// TwinCAT 3 PLC project Untitled1
// ProgramVersion: 3.1.4024.0
// libraries:
//   Tc2_Math, * (Beckhoff Automation GmbH)
//   Tc2_Standard, * (Beckhoff Automation GmbH)
//   Tc2_System, * (Beckhoff Automation GmbH)
//   Tc2_Utilities, * (Beckhoff Automation GmbH)
//   Tc3_CM, * (Beckhoff Automation GmbH)
//   Tc3_CM_Base, * (Beckhoff Automation GmbH)
//   Tc3_IotBase, * (Beckhoff Automation GmbH)
//   Tc3_JsonXml, * (Beckhoff Automation GmbH)
//   Tc3_Module, * (Beckhoff Automation GmbH)
//   Tc3_MultiArray, * (Beckhoff Automation GmbH)
// project tree:
//   / CM_Process_Task.TcTTO, HTTP_Task.TcTTO, PlcTask.TcTTO
//   DUTs/Error Monitoring/ ST_HRErrHist.TcDUT, E_TalkToGateway_Err.TcDUT
//   DUTs/ E_AnalysisIDs.TcDUT, E_IsoClass.TcDUT, E_RequestType.TcTLEO, ST_ReceivedData.TcDUT
//   DUTs/Function Generator/ E_FunctionType.TcDUT
//   FUBs/ FB_Flash.TcPOU, FB_FunctionGenerator.TcPOU, FB_FunctionGenerator_1.TcPOU, FB_HRErrHist.TcPOU
//   GVLs/ GLOBAL.TcGVL, GVL_Const.TcGVL
//   POUs/CM_Collection/ CM_SensorWorks_Sensor1.TcPOU, CM_SensorWorks_Sensor2.TcPOU, CM_Sim.TcPOU
//   POUs/CM_Processing/ CM_SensorWorks_Sensor1ISO.TcPOU, CM_SensorWorks_Sensor2ISO.TcPOU, CM_Sim_ISO.TcPOU
//   POUs/HTTP/ FB_RequestToGateway.TcPOU, FB_TalkToGateway.TcPOU, GetDataFromSensorWorksHTTP.TcPOU
//   POUs/ MAIN.TcPOU
// real-time tasks:
//   TASK PlcTask: cycle T#25000us, priority 10, ADS port 350
//   TASK CM_Process_Task: cycle T#50000us, priority 4, ADS port 351
//   TASK HTTP_Task: cycle T#500ms, priority 20, ADS port 352

CONFIGURATION Untitled1
    RESOURCE PLC ON TwinCAT3
        TASK CM_Process_Task(INTERVAL := T#50000us, PRIORITY := 4);
        TASK HTTP_Task(INTERVAL := T#500ms, PRIORITY := 20);
        TASK PlcTask(INTERVAL := T#25000us, PRIORITY := 10);
        PROGRAM CM_Sim_ISO WITH CM_Process_Task : CM_Sim_ISO;
        PROGRAM CM_SensorWorks_Sensor1ISO WITH CM_Process_Task : CM_SensorWorks_Sensor1ISO;
        PROGRAM CM_SensorWorks_Sensor2ISO WITH CM_Process_Task : CM_SensorWorks_Sensor2ISO;
        PROGRAM MAIN WITH PlcTask : MAIN;
    END_RESOURCE
END_CONFIGURATION

// ---- DUTs/Error Monitoring/ST_HRErrHist.TcDUT
TYPE ST_HRErrHist :
STRUCT
{attribute 'displaymode':='hex'}
	hrErrCode	: HRESULT;
	sErrSource	: STRING(63);
	nErrCount	: UDINT;
END_STRUCT
END_TYPE

// ---- DUTs/Error Monitoring/E_TalkToGateway_Err.TcDUT

TYPE
    E_TalkToGateway_Err :
    (
        e_NoIPAddress           := 10,
        e_NoPortNumber          := 20,
        e_NoDeviceID            := 30,
        e_DeviceIDOutsideLimits := 31,
        e_DeviceIDNotFound      := 32,
		e_JSONRequestError		:= 40
        );
END_TYPE

// ---- DUTs/E_AnalysisIDs.TcDUT
TYPE
    E_AnalysisIDs :
    (
        (* analysis chain *)
        eID_SimSource := 1,
        eID_SimISO,
        eID_SimSinkISO,
        eID_SimSpectrumCh1,
        eID_SimSpectrumCh2,
        eID_SimSinkSpectrumCh1,
        eID_SimSinkSpectrumCh2,
        eID_SensorWorksSource,
        eID_SensorWorksISO,
        eID_SensorWorksSpectrum,
        eID_SensorWorksSinkISO,
        eID_SensorWorkSinkSpectrum,
        eID_SW_Source_Device_1,
        eID_SW_ISO_Device_1,
        eID_SW_Sink_Device_1,
        eID_SW_Source_Device_2,
        eID_SW_ISO_Device_2,
        eID_SW_Sink_Device_2
    ) UDINT;
END_TYPE

// ---- DUTs/E_IsoClass.TcDUT
(* ISO Classes *)
{attribute 'qualified_only'}
TYPE E_IsoClass :
(
	A := 1,
	B,
	C,
	D
) UDINT;
END_TYPE

// ---- DUTs/E_RequestType.TcTLEO

TYPE E_RequestType :
(
	eIdle,
	eSampleRate,
	eTraceLen,
	eMode,
	eRequestSend,
	eViewRequest, // ✅ Add this line
	eGetData,
	eProcess,
	eERROR
);
END_TYPE

// ---- DUTs/Function Generator/E_FunctionType.TcDUT
{attribute 'qualified_only'}
TYPE E_FunctionType :
(
	Sine,		// typical for vibrations originating from rotating machine
	Square,		// mixed sine signals good for analyzing spectrum
	Pulse,		// mixed sine signals good for analyzing spectrum
	Triangular,	// mixed sine signals good for analyzing spectrum
	Sawtooth,	// ramp-type vibrations, continuously increasing
	AM			// amplitude modulation: typical for vibrations originating from gear-tooth failure or bearing faults
);
END_TYPE

// ---- DUTs/ST_ReceivedData.TcDUT
TYPE ST_ReceivedData :
STRUCT
	uuid			: STRING;
	blename			: STRING;
	name			: STRING;
	id				: STRING;
	timestamp		: STRING;
	value 			: ARRAY[0..512] OF DINT;
	value_y			: ARRAY[0..512] OF DINT;
	value_z			: ARRAY[0..512] OF DINT;
	rate			: DINT;
	trace			: DINT;
	count			: DINT;
	gain			: DINT;
	calibration		: LREAL;
	calibration_y	: LREAL;
	calibration_z	: LREAL;
	temperature		: LREAL;
	battery			: LREAL;
	axes			: LREAL;
	mux_axis		: LREAL;
	measured_rate	: LREAL;
	
END_STRUCT
END_TYPE

// ---- GVLs/GLOBAL.TcGVL
{attribute 'qualified_only'}
VAR_GLOBAL
    {attribute 'TcAnalytics'}
    aSimBuffer : ARRAY[1..GVL_Const.cChannels] OF ARRAY[1..GVL_Const.cOversamples] OF LREAL;
    aSimRMSResult         : ARRAY[1..GVL_Const.cChannels] OF ARRAY[1..GVL_Const.cResult_Length] OF LREAL;
    aSimSpectrumCh1Result : ARRAY[1..(GVL_Const.cFFTLength / 2 + 1)] OF LREAL;
    aSimSpectrumCh2Result : ARRAY[1..(GVL_Const.cFFTLength / 2 + 1)] OF LREAL;

	(****** Sensor Works ******)
    stSensorWorksHTTPSensorData : ARRAY[1..GVL_Const.cMaxVibrationDevices] OF ST_ReceivedData; // Data from the devices
    aSensorWorksHTTPInput    : ARRAY[1..GVL_Const.cMaxVibrationDevices] OF ARRAY[1..GVL_Const.cSensorPacket] OF LREAL; // Scaled data to input into vibration FuBs
    aSensorWorkISOHTTPResult : ARRAY[1..GVL_Const.cMaxVibrationDevices] OF ARRAY[1..GVL_Const.cResult_Length] OF LREAL; // Output values from Sink

    strTimeStamp : STRING;
    strIPAddress : STRING := '192.168.4.44';
	//strIPAddress : STRING := '192.168.216.148';
	//strDeviceID  : ARRAY[1..GVL_Const.cMaxVibrationDevices] OF STRING := ['d5:d0:f9:30:83:d7'];
	
	strDeviceID  : ARRAY[1..GVL_Const.cMaxVibrationDevices] OF STRING := ['fa:e2:ad:e2:8d:99', 'd5:d0:f9:30:83:d7'];
    nPortNumber  : UINT := 8080;
	
	bCommError : BOOL := FALSE;     // Qin
//	fbCommErrHist : FB_ErrHist;
    bIsProcessingRequest : BOOL := FALSE;
    strLastRequestOutput : STRING(255);
	
	iAnalueIn1 AT %I* : INT;  // Qin
	Sensor1Ch1AccRMSiAnalueIn2 AT %I* : INT;
	
Sensor1Ch1AccRMS : ARRAY[1..28] OF REAL := [
    37.0, 15.0, 10.0, 23.0, 17.0, 21.0, 23.0, 17.0,
    24.0, 18.0, 3.0, 18.0, 38.0, 29.0, 11.0, 0.0,
    7.0, 20.0, 8.0, 7.0, 24.0, 9.0, 1.0, 28.0,
    29.0, 19.0, 30.0, 28.0
];




END_VAR

// ---- GVLs/GVL_Const.TcGVL
{attribute 'qualified_only'}
VAR_GLOBAL CONSTANT

    cFSample      : UDINT := 10000; // 1ms task with 10 oversamples = 10kHz
    cMaxBins      : UDINT := 100;
    cMaxQuantiles : UDINT := 2;
    cMaxClasses   : UDINT := 3; // Normal, Warning, Alarm		

    // define frequency interval according to ISO 10816-3
    // e.g. 10 .. 1000 Hz for rotating speed over 600r/min
    cfLowerFrequencyLimit : UDINT := 10;
    cfUpperFrequencyLimit : UDINT := 1000;

    // Parameters for RMS calculation
    cOrderRMS      : UDINT := 2;             // ISO 10816-3 requires velocity and displacement, if measured using accelerometer we need to integrate 2 times
    cChannels      : UDINT := 2;             // ISO 10816-3 says 2 orthogonal sensors per measurement location-> 2 channels
    cResult_Length : UDINT := cOrderRMS + 1; // nOrder+1
    cSensorSampleChannels
        : UDINT := 1;

    // Classes according to ISO:
    // machine, elasticty, value
    cISOClassDef_Velocity : ARRAY[1..2, 1..2, 1..3] OF LREAL := [0.0023,
                                                                 0.0045,
                                                                 0.0071,
                                                                 0.0035,
                                                                 0.0071,
                                                                 0.011,
                                                                 0.0014,
                                                                 0.0028,
                                                                 0.0045,
                                                                 0.0023,
                                                                 0.0045,
                                                                 0.0071];
    cISOClassDef_Displ : ARRAY[1..2, 1..2, 1..3] OF LREAL := [2.9E-05,
                                                              5.7E-05,
                                                              9E-05,
                                                              4.5E-05,
                                                              9E-05,
                                                              0.00014,
                                                              2.2E-05,
                                                              4.5E-05,
                                                              7.1E-05,
                                                              3.7E-05,
                                                              7.1E-05,
                                                              0.000113];

    // optional constants if real sensors are applied
    cGravitationalAcc : LREAL := 9.81;  // 1 g approx 9.81 m/s^2 -> physical constant
    cSensitivity      : LREAL := 0.01;  // [in Volts/g] depends on sensor used in application, e.g. 10 mV/g
    cMeasurementRange : LREAL := 5;     // +-5 Volts (EL3632)
    cResolution       : LREAL := 32768; // 2^15 (15 bits resolution + 1 bit sign) (EL3632)
    cScale            : LREAL := cMeasurementRange * cGravitationalAcc / (cSensitivity * cResolution);

    // Application ConMon constants
    cSensorPacket          : UDINT                 := 512; // Number of samples in the packet incoming from the sensor	
    cSensorSampleRate      : UDINT                 := 256;
    cOversamples           : UDINT                 := 10;                             // number of oversamples
    cMaxChannels           : UDINT                 := 5;                              // number of data channels
    cWindowType            : E_CM_WindowType       := E_CM_WindowType.eCM_HannWindow; // window type for analysis
    cWindowParameters      : T_CM_WindowParameters := [0, 0, 0, 0, 0];                // window parameters
    cWindowLength          : UDINT                 := 3200;                           // length of signal window 
    cOverlap               : UDINT                 := 1600;                           // recommended buffer overlap
    cBufferLength          : UDINT                 := cWindowLength - cOverlap;       // internal buffer size with 50% overlapping	                                            						
    cFFTLength             : UDINT                 := 4096;                           // length of FFT for mag. spectrum
    cFFTResult             : UDINT                 := 2049;                           // result of mag. spectrum (cFFTLength/2+1)
    cBufferLength_Spectrum : UDINT                 := 1600;                           // buffer size due to 50% overlap

    //Alarm Constants
    cMax_Alarms : UINT := 99;

    // Device Constants
    cMaxVibrationDevices : UINT := 10;

END_VAR

// ---- POUs/CM_Processing/CM_Sim_ISO.TcPOU
PROGRAM CM_Sim_ISO
VAR CONSTANT
		cInitIntRMS 	: ST_CM_IntegratedRMS_InitPars   := (	nFFT_Length := GVL_Const.cFFTLength, 
															nWindowLength := GVL_Const.cWindowLength,
															fSampleRate := GVL_Const.cFSample,
		 													fLowerFrequencyLimit := GVL_Const.cfLowerFrequencyLimit,
															fUpperFrequencyLimit := GVL_Const.cfUpperFrequencyLimit,
															nOrder := GVL_Const.cOrderRMS,
															nChannels := GVL_Const.cChannels,                        
															eWindowType := E_CM_WindowType.eCM_HannWindow, 
															bTransformToDecibel:= FALSE);		

END_VAR
VAR
		fbRMS				: FB_CMA_IntegratedRMS  	  :=(	stInitPars := cInitIntRMS, 
															nOwnID := eID_SimISO, 
															aDestIDs := [eID_SimSinkISO] );

	fbErrHist			: FB_HRErrHist; // error monitoring


END_VAR

// Call RMS
fbRMS.Call();

IF fbRMS.bError THEN
	fbErrHist.AddError(bErr:=TRUE, hrErrCode:=fbRMS.hrErrorCode, sErrSource:='CM_Sim_ISO.fbRMS'); // error monitoring
	// ToDo: if error
END_IF

END_PROGRAM

// ---- FUBs/FB_HRErrHist.TcPOU
FUNCTION_BLOCK FB_HRErrHist
(* v1.10
build up an error history consisting of two arrays and one index.
The index shows the actual array position. The last error id and the count for this id are saved in the arrays.
If an error id is the same as the previous input error the counter is increased. Otherwise the index is increased.
*)
VAR_INPUT
	bEdgeDetect	: BOOL;	(* FALSE: every input(bErr) is processed; TRUE: only rising edge of input is processed *)
END_VAR
VAR_OUTPUT
	nErrSum		: UINT;
	nErrIdx		: UINT; // error list index of last occured error (max. cHistLen)
	aErrList	: ARRAY[1..cHistLen] OF ST_HRErrHist;
END_VAR

VAR
	bNewErr		: BOOL;
	fbErrTrig	: R_TRIG;
END_VAR
VAR CONSTANT
	cHistLen	: UINT := 100;
END_VAR

METHOD AddError
VAR_INPUT
	bErr		: BOOL;
	hrErrCode	: HRESULT;
	sErrSource	: STRING(63);
END_VAR
fbErrTrig(CLK:=bErr);
IF bEdgeDetect THEN
	bNewErr := fbErrTrig.Q;
ELSE
	bNewErr := bErr;
END_IF

IF bNewErr THEN
	nErrSum := nErrSum + 1;
	IF nErrIdx < cHistLen THEN
		IF nErrIdx = 0 THEN
			nErrIdx	:= nErrIdx + 1;
		ELSIF aErrList[nErrIdx].hrErrCode <> hrErrCode OR aErrList[nErrIdx].sErrSource <> sErrSource THEN
			nErrIdx	:= nErrIdx + 1;
		END_IF
		aErrList[nErrIdx].hrErrCode := hrErrCode;
		aErrList[nErrIdx].sErrSource := sErrSource;
		aErrList[nErrIdx].nErrCount := aErrList[nErrIdx].nErrCount + 1;
	END_IF
END_IF
END_METHOD

METHOD Reset
VAR_INPUT
END_VAR
nErrSum := 0;
nErrIdx := 0;
MEMSET(ADR(aErrList),0,SIZEOF(aErrList));
END_METHOD

END_FUNCTION_BLOCK

// ---- POUs/CM_Processing/CM_SensorWorks_Sensor1ISO.TcPOU
PROGRAM CM_SensorWorks_Sensor1ISO

VAR CONSTANT
		cInitIntRMS 	: ST_CM_IntegratedRMS_InitPars   := (	nFFT_Length := GVL_Const.cSensorPacket, 
															nWindowLength := GVL_Const.cSensorPacket,
															fSampleRate := GVL_Const.cSensorSampleRate, // packets per second, sample time is 2s
		 													fLowerFrequencyLimit := 10,
															fUpperFrequencyLimit := 100,	// needs to be less than half of the sample rate
															nMaxBands:= 1, 										
															nOrder := 2,
															nChannels := 1,                        
															eWindowType := E_CM_WindowType.eCM_HannWindow,
															nOverlap:= 0, 
															bTransformToDecibel:= FALSE);

END_VAR

VAR
	fbRMS				: FB_CMA_IntegratedRMS  	  :=(	stInitPars := cInitIntRMS, 
															nOwnID := eID_SW_ISO_Device_1, 
															aDestIDs := [eID_SW_Sink_Device_1],
															nResultBuffers:= 4);
	
	bInit: BOOL := TRUE;														
	aBands				: ARRAY [1..2] OF LREAL := [10.0, 100.0];
	hResInit			:  HRESULT;										

	fbErrHist			: FB_HRErrHist; // error monitoring

END_VAR

IF bInit THEN
	hResInit := fbRms.Configure(pArg:= ADR(aBands), nArgSize:= SIZEOF(aBands));
	bInit := FALSE;
END_IF

// Call RMS
fbRMS.Call();

IF fbRMS.bError THEN
	fbErrHist.AddError(bErr:=TRUE, hrErrCode:=fbRMS.hrErrorCode, sErrSource:='CM_SensorWorks_Sensor1ISO.fbRMS'); // error monitoring
	// ToDo: if error
END_IF

END_PROGRAM

// ---- POUs/CM_Processing/CM_SensorWorks_Sensor2ISO.TcPOU
PROGRAM CM_SensorWorks_Sensor2ISO

VAR CONSTANT
    cInitIntRMS : ST_CM_IntegratedRMS_InitPars := (nFFT_Length          := GVL_Const.cSensorPacket,
                                                   nWindowLength        := GVL_Const.cSensorPacket,
                                                   fSampleRate          := GVL_Const.cSensorSampleRate, // packets per second, sample time is 2s
                                                   fLowerFrequencyLimit := 10,
                                                   fUpperFrequencyLimit := 100, // needs to be less than half of the sample rate
                                                   nMaxBands            := 1,
                                                   nOrder               := 2,
                                                   nChannels            := 1,
                                                   eWindowType          := E_CM_WindowType.eCM_HannWindow,
                                                   nOverlap             := 0,
                                                   bTransformToDecibel  := FALSE);

END_VAR

VAR
    fbRMS : FB_CMA_IntegratedRMS := (stInitPars     := cInitIntRMS,
                                     nOwnID         := eID_SW_ISO_Device_2,
                                     aDestIDs       := [eID_SW_Sink_Device_2],
                                     nResultBuffers := 4);

    bInit    : BOOL                 := TRUE;
    aBands   : ARRAY[1..2] OF LREAL := [10.0, 100.0];
    hResInit : HRESULT;

    fbErrHist : FB_HRErrHist; // error monitoring

END_VAR

IF bInit THEN
    hResInit := fbRms.Configure(pArg := ADR(aBands), nArgSize := SIZEOF(aBands));
    bInit    := FALSE;
END_IF

// Call RMS
fbRMS.Call();

IF fbRMS.bError THEN
    fbErrHist.AddError(bErr := TRUE, hrErrCode := fbRMS.hrErrorCode, sErrSource := 'CM_SensorWorks_Sensor2ISO.fbRMS'); // error monitoring
    // ToDo: if error
END_IF

END_PROGRAM

// ---- POUs/MAIN.TcPOU
PROGRAM MAIN
VAR
	// Task Vars
	nChannel: UDINT;
	fbFunctionGenerator1	: FB_FunctionGenerator;		// Signal Generator, ch1
	fbFunctionGenerator2	: FB_FunctionGenerator;		// Signal Generator, ch2
	fSetFrequency1			: LREAL := 400;		        // Hz
	fSetAmplitude1			: LREAL := 4;		        // peak amplitude of sin signal [m/s^2]
	fSetFrequency2			: LREAL := 35;		        // Hz
	fSetAmplitude2			: LREAL := 4;		        // peak amplitude of sin signal	[m/s^2]	
	
	bAddDisturbance			: BOOL;											// add fault
	fbDisturbance1			: FB_FunctionGenerator;							// fault simulator
	fDistAmplitude1			: LREAL	:= 5;									// fault amplitude
	fDistFrequency1			: LREAL	:= 200;									// fault frequency (recurring)
	fbDisturbance2			: FB_FunctionGenerator;							// fault simulator
	fDistAmplitude2			: LREAL	:= 2;									// fault amplitude
	fDistFrequency2			: LREAL	:= 100;									// fault frequency (recurring)

	eDistFunction			: E_FunctionType :=  E_FunctionType.Square;	// fault shape
	aDisturbance			: ARRAY[1..GVL_Const.cChannels] OF ARRAY[1..GVL_Const.cOversamples] OF LREAL;

	fbRand					: DRAND;				 	
	fRandomNumber			: LREAL;	
	fVar					: LREAL := 0.38;

	nSample					: UDINT;

	fbTalkToGateway			: FB_TalkToGateway;

END_VAR

VAR   //Qin
    fbSendEdge : R_TRIG;

    bTriggerSend : BOOL := FALSE;
    bStartPulse  : BOOL := TRUE;

    fbHttpClient : FB_IotHttpClient;

   // strRawJson : STRING(8191);

    bBusy   : BOOL;
    bError  : BOOL;
END_VAR


// Simulated frequency generation
fbFunctionGenerator1(fFrequency := fSetFrequency1,
                     fAmplitude := fSetAmplitude1,
                     eFunction  := E_FunctionType.Sine,
                     aSignal    := GLOBAL.aSimBuffer[1]);

fbFunctionGenerator2(fFrequency := fSetFrequency2,
                     fAmplitude := fSetAmplitude2,
                     eFunction  := E_FunctionType.Sine,
                     aSignal    := GLOBAL.aSimBuffer[2]);

IF bAddDisturbance THEN
    // Random number generator
    fbRand(Seed := 1000, Num => fRandomNumber);
    (* Disturbance signal *)
    fbDisturbance1(bEnable    := TRUE,
                   fAmplitude := fDistAmplitude1,
                   fFrequency := fDistFrequency1,
                   fOffset    := 0,
                   nDutyCycle := 2,
                   eFunction  := eDistFunction,
                   aSignal    := aDisturbance[1]);

    fbDisturbance2(bEnable    := TRUE,
                   fAmplitude := fDistAmplitude2,
                   fFrequency := fDistFrequency2,
                   fOffset    := 0,
                   nDutyCycle := 2,
                   eFunction  := eDistFunction,
                   aSignal    := aDisturbance[2]);

    FOR nChannel := 1 TO GVL_Const.cChannels DO
        // Input signal with disturbance
        FOR nSample := 1 TO GVL_Const.cOversamples DO
            GLOBAL.aSimBuffer[nChannel][nSample] := GLOBAL.aSimBuffer[nChannel][nSample] + fRandomNumber * aDisturbance[nChannel][nSample];
        END_FOR
    END_FOR

END_IF

// Statically writing devices for ease during testing
//GLOBAL.strDeviceID[1] := 'e0:f6:fd:c4:e3:08';
//GLOBAL.strDeviceID[2] := 'd5:d0:f9:30:83:d7';

// Instance call to FB_TalkToGateway
fbTalkToGateway(
    strIPAddress        := GLOBAL.strIPAddress,
    nPortNumber         := GLOBAL.nPortNumber,
    strDeviceID         := GLOBAL.strDeviceID,
    bStopConnection     :=,                                  // TODO: Set logic to stop the connection when needed.  
    bResetError         := FALSE,                                  // TODO: Link to a button or watchdog to reset error
    bSendRequest        := ,                                   // Should be controlled by a trigger condition
    eRequestType := E_RequestType.eViewRequest,
	//eRequestType        := E_RequestType.eGetData,              // Replace with actual enum value as needed
    iRequestDeviceIndex := 1,                                      // Index of the device to talk to (1 or 2)
    tPollTime           := T#1S,
    bError              => GLOBAL.bCommError,                      // Assign your error flag
//    fbErrHist           => GLOBAL.fbCommErrHist,                   // Optional: instantiate this function block globally
    aDeviceResponse     => GLOBAL.stSensorWorksHTTPSensorData,    // Structure to receive sensor data
    strRequestOutput    => GLOBAL.strLastRequestOutput,           // Optional: use to log or debug request payloads
    bProcessingRequest  => GLOBAL.bIsProcessingRequest            // Track request state
);


// this block Qin
IF bStartPulse THEN
    bTriggerSend := TRUE;
    bStartPulse := FALSE;
ELSE
    bTriggerSend := FALSE;
END_IF


// Detect rising edge
fbSendEdge(CLK := bTriggerSend);

// Call your FB   //Qin
(*
fbGetDataFromSensor(
    bSend := fbSendEdge.Q,
    strRequest := '/device/d5:d0:f9:30:83:d7/cache/latest',   // Qin
    bErrorReset := FALSE,
    fbClient := fbHttpClient,
    bBusy => bBusy,
    bError => bError
);
*)

// View raw content
// strRawJson := fbGetDataFromSensor.sContent;   //Qin


// Cyclic Program Calls
CM_Sim();
CM_SensorWorks_Sensor1();
CM_SensorWorks_Sensor2();

END_PROGRAM

// ---- FUBs/FB_FunctionGenerator.TcPOU
// generates a signal build up by the specified function type. v1.6
FUNCTION_BLOCK FB_FunctionGenerator
VAR_INPUT
	bEnable		: BOOL 	:= TRUE;	// set TRUE to generate the specified signal; set FALSE to reset the signal buffer
	fFrequency	: LREAL := 1000;	// in [Hz]
	fAmplitude	: LREAL := 1;
	fOffset		: LREAL	:= 0;	
	nDutyCycle	: UINT 	:= 50;		// in [%] (for pulse function)
	eFunction	: E_FunctionType := E_FunctionType.Sine;	
END_VAR
VAR_IN_OUT
	aSignal		: ARRAY[1..GVL_Const.cOversamples] OF LREAL;
END_VAR
VAR_OUTPUT
	bError		: BOOL;
END_VAR

VAR
	bInit						: BOOL := TRUE;
	fbGetTaskIdx				: GETCURTASKINDEX;
	
	fLastFrequency				: LREAL;		// in [Hz]
	fLastAmplitude				: LREAL;
	fLastOffset					: LREAL;
	nLastDutyCycle				: UINT;
	eLastFunction				: E_FunctionType;
	
	nSamples					: UDINT;
	fCycleTime					: LREAL;		// in [s]
	fDelta						: LREAL;		// amplitude delta per sample
	fPhase						: LREAL;		// in [°]
	nSign						: INT := 1;		// 1 or -1
	fLastSignalValue			: LREAL;		// amplitude
	fPeriod						: LREAL;		// in [s]
	fAngularIncrement			: LREAL;		// in [°]
	fAngularIncrementPerCycle	: LREAL;		// in [°]
	fAngularIncrementPerSample	: LREAL;		// in [°]
	(* for modulated signal (carrier signal without offset) *)
	fCarrierFrequency					: LREAL := 500;	// in [Hz] (sine)
	fCarrierAmplitude					: LREAL := 1;
	fCarrierPeriod						: LREAL;		// in [s]
	fCarrierAngularIncrement			: LREAL;		// in [°]
	fCarrierAngularIncrementPerCycle	: LREAL;		// in [°]
	fCarrierAngularIncrementPerSample	: LREAL;		// in [°]
				
END_VAR

IF bEnable THEN
	IF fLastFrequency <> fFrequency THEN
		bInit := TRUE; // For automatic initializing
		fLastFrequency := fFrequency;
	END_IF
	IF fLastAmplitude <> fAmplitude THEN
		bInit := TRUE; // For automatic initializing
		fLastAmplitude := fAmplitude;
	END_IF
	IF fLastOffset <> fOffset THEN
		bInit := TRUE; // For automatic initializing
		fLastOffset := fOffset;
	END_IF
	IF nLastDutyCycle <> nDutyCycle THEN
		bInit := TRUE; // For automatic initializing
		nLastDutyCycle := nDutyCycle;
	END_IF
	IF eLastFunction <> eFunction THEN
		bInit := TRUE; // For automatic initializing
		eLastFunction := eFunction;
	END_IF
	IF bInit THEN
		// Get task info	
		fbGetTaskIdx();
		fCycleTime := UDINT_TO_LREAL(TwinCAT_SystemInfoVarList._TaskInfo[fbGetTaskIdx.index].CycleTime) (*100ns*) / (10.0 * 1000.0 * 1000.0);	
		fLastSignalValue := 0;
		nSign := 1;
		fAngularIncrement := 0;
		// Flush out old data
		MEMSET(ADR(aSignal), 0, SIZEOF(aSignal));
		IF fFrequency > 0 AND fCycleTime > 0 THEN		
			// Calculate period, increments per plc cycle, increment per oversample
			IF GVL_Const.cOversamples > 0 THEN			
				IF eFunction = E_FunctionType.Sine THEN
					fPeriod := 1/fFrequency;
					fAngularIncrementPerCycle := 360*(fCycleTime/fPeriod);
					fAngularIncrementPerSample := fAngularIncrementPerCycle/GVL_Const.cOversamples;
					// no phase adjustment
					bInit := FALSE;	
				ELSIF eFunction = E_FunctionType.Square	THEN
					fPeriod := 1/fFrequency;
					fAngularIncrementPerCycle  := 360*(fCycleTime/fPeriod);
					fAngularIncrementPerSample := fAngularIncrementPerCycle/GVL_Const.cOversamples;
					fPhase := 0.5*360;
					bInit := FALSE;
				ELSIF eFunction = E_FunctionType.Pulse THEN
					fPeriod := 1/fFrequency;
					fAngularIncrementPerCycle  := 360*(fCycleTime/fPeriod);
					fAngularIncrementPerSample := fAngularIncrementPerCycle/GVL_Const.cOversamples;
					IF nDutyCycle > 100 THEN
						nDutyCycle := 100;
					END_IF
					fPhase := (UDINT_TO_LREAL(nDutyCycle)/100)*360;
					bInit := FALSE;					
				ELSIF eFunction = E_FunctionType.Triangular THEN
					fPeriod := 1/fFrequency;				
					fAngularIncrementPerCycle  := 360*(fCycleTime/fPeriod);
					fAngularIncrementPerSample := fAngularIncrementPerCycle/GVL_Const.cOversamples;
					fPhase := 0.5*360; 
					fDelta := 4*(fAmplitude/(360/fAngularIncrementPerSample));				
					bInit := FALSE;
				ELSIF eFunction = E_FunctionType.Sawtooth THEN
					fPeriod := 1/fFrequency;			
					fAngularIncrementPerCycle  := 360*(fCycleTime/fPeriod);		
					fAngularIncrementPerSample := fAngularIncrementPerCycle/GVL_Const.cOversamples;
					fDelta := fAmplitude/(360/fAngularIncrementPerSample);
					bInit := FALSE;
				ELSIF eFunction = E_FunctionType.AM THEN
					fPeriod := 1/fFrequency;
					fAngularIncrementPerCycle := 360*(fCycleTime/fPeriod);
					fAngularIncrementPerSample := fAngularIncrementPerCycle/GVL_Const.cOversamples;
					// no phase adjustment
					fCarrierPeriod := 1/fCarrierFrequency;
					fCarrierAngularIncrementPerCycle := 360*(fCycleTime/fCarrierPeriod);
					fCarrierAngularIncrementPerSample := fCarrierAngularIncrementPerCycle/GVL_Const.cOversamples;				
					// no phase adjustment	
					bInit := FALSE;
				ELSE
					bError := TRUE;	
				END_IF
			ELSE
				bError := TRUE;
			END_IF
		ELSE
			bError := TRUE;
		END_IF
	END_IF
	
	// Enable function generator
	IF NOT bError THEN		
		CASE eFunction OF		
			// sine: typical for vibrations originating from rotating machine
			E_FunctionType.Sine: Sine();
			
			// square: mixed sine signals good for analyzing spectrum				
			E_FunctionType.Square: Square();
			
			// pulse: mixed sine signals good for analyzing spectrum				
			E_FunctionType.Pulse: Pulse();
	
			// sawtooth: ramp-type vibrations, continuously increasing			
			E_FunctionType.Sawtooth: Sawtooth();
		
			// triangular: mixed sine signals good for analyzing spectrum
			E_FunctionType.Triangular: Triangular();
		
			// amplitude modulation: typical for vibrations originating from gear-tooth failure or bearing faults
			// Carrier signal with own frequency and amplitude		
			E_FunctionType.AM: AM();				
		END_CASE
	END_IF
ELSE
	// Flush out old data
	MEMSET(ADR(aSignal), 0, SIZEOF(aSignal));
	
	bInit := TRUE;
	bError := FALSE;
END_IF

METHOD PRIVATE AM
VAR_INPUT
END_VAR
{warning disable C0371}

FOR nSamples := 1 TO GVL_Const.cOversamples DO
	// base signal * carrier signal
	aSignal[nSamples] := ( fAmplitude*SIN(2*PI*(fAngularIncrement+(nSamples-1)*fAngularIncrementPerSample)/360) + fOffset )
							* ( fCarrierAmplitude*SIN(2*PI*(fCarrierAngularIncrement+(nSamples-1)*fCarrierAngularIncrementPerSample)/360) );
END_FOR
// Increment angular positions
fAngularIncrement := fAngularIncrement + fAngularIncrementPerCycle;
fCarrierAngularIncrement := fCarrierAngularIncrement + fCarrierAngularIncrementPerCycle;

{warning restore C0371}
END_METHOD

METHOD PRIVATE Pulse
VAR_INPUT
END_VAR
{warning disable C0371}

FOR nSamples := 1 TO GVL_Const.cOversamples DO
	// For pulse wave (unequal phases)
	IF (fAngularIncrement >= 360) THEN
		fAngularIncrement := fAngularIncrement - DINT_TO_LREAL(LREAL_TO_DINT(fAngularIncrement/360))*360;
		// or with Tc2_Math library: fAngularIncrement := LMOD(fAngularIncrement,360);
	END_IF
	IF (fAngularIncrement < fPhase) THEN
		nSign := 1;		
	ELSIF (fAngularIncrement >= fPhase) THEN
		nSign := 0;
	END_IF
	fAngularIncrement := fAngularIncrement + fAngularIncrementPerSample;
	
	aSignal[nSamples] := nSign*fAmplitude;
	
	aSignal[nSamples] := aSignal[nSamples] + fOffset;
END_FOR

{warning restore C0371}
END_METHOD

METHOD PRIVATE Sawtooth
VAR_INPUT
END_VAR
{warning disable C0371}

FOR nSamples := 1 TO GVL_Const.cOversamples DO
	// For sawtooth wave (equal phase = period/2)
	IF (fAngularIncrement >= 360) THEN
		fAngularIncrement := fAngularIncrement - DINT_TO_LREAL(LREAL_TO_DINT(fAngularIncrement/360))*360;
		// or with Tc2_Math library: fAngularIncrement := LMOD(fAngularIncrement,360);
		fLastSignalValue := fLastSignalValue -fAmplitude;
	END_IF
	fAngularIncrement := fAngularIncrement + fAngularIncrementPerSample;

	aSignal[nSamples] := fLastSignalValue + fDelta;

	// Store last sample
	fLastSignalValue := aSignal[nSamples];
	
	aSignal[nSamples] := aSignal[nSamples] + fOffset;					
END_FOR	

{warning restore C0371}
END_METHOD

METHOD PRIVATE Sine
VAR_INPUT
END_VAR
{warning disable C0371}

FOR nSamples := 1 TO GVL_Const.cOversamples DO
	aSignal[nSamples] := fAmplitude*SIN(2*PI*(fAngularIncrement+(nSamples-1)*fAngularIncrementPerSample)/360);

	aSignal[nSamples] := aSignal[nSamples] + fOffset;
END_FOR

// Increment angular position
fAngularIncrement := fAngularIncrement + fAngularIncrementPerCycle;

{warning restore C0371}
END_METHOD

METHOD PRIVATE Square
VAR_INPUT
END_VAR
{warning disable C0371}

FOR nSamples := 1 TO GVL_Const.cOversamples DO
	// For square wave (equal phase = period/2)
	IF (fAngularIncrement >= 360) THEN
		fAngularIncrement := fAngularIncrement - DINT_TO_LREAL(LREAL_TO_DINT(fAngularIncrement/360))*360;
		// or with Tc2_Math library: fAngularIncrement := LMOD(fAngularIncrement,360);
	END_IF
	IF (fAngularIncrement < fPhase) THEN
		nSign := 1;
	ELSIF (fAngularIncrement >= fPhase) THEN
		nSign := -1;
	END_IF
	fAngularIncrement := fAngularIncrement + fAngularIncrementPerSample;
	
	aSignal[nSamples] := nSign*fAmplitude;
	
	aSignal[nSamples] := aSignal[nSamples] + fOffset;
END_FOR

{warning restore C0371}
END_METHOD

METHOD PRIVATE Triangular
VAR_INPUT
END_VAR
{warning disable C0371}

FOR nSamples := 1 TO GVL_Const.cOversamples DO
	IF (fAngularIncrement >= 360) THEN
		fAngularIncrement := fAngularIncrement - DINT_TO_LREAL(LREAL_TO_DINT(fAngularIncrement/360))*360;
		// or with Tc2_Math library: fAngularIncrement := LMOD(fAngularIncrement,360);
	END_IF
	// Negative delta -> Positive delta
	IF fAngularIncrement < fPhase/2 THEN	
		nSign := 1;		
	ELSIF fAngularIncrement >= fPhase/2 AND fAngularIncrement < 3*fPhase/2 THEN
		nSign := -1;
	ELSIF fAngularIncrement >= 3*fPhase/2 THEN
		nSign := 1;	
	END_IF
	fAngularIncrement := fAngularIncrement + fAngularIncrementPerSample;
	
	aSignal[nSamples] := fLastSignalValue + nSign*fDelta;
	IF aSignal[nSamples] > fAmplitude THEN
		aSignal[nSamples] := aSignal[nSamples] - 2*(aSignal[nSamples]-fAmplitude);
	ELSIF aSignal[nSamples] < (-1)*fAmplitude THEN
		aSignal[nSamples] := aSignal[nSamples] - 2*(aSignal[nSamples]+fAmplitude);
	END_IF
	
	// Store last sample
	fLastSignalValue := aSignal[nSamples];		
	
	aSignal[nSamples] := aSignal[nSamples] + fOffset;
END_FOR

{warning restore C0371}
END_METHOD

END_FUNCTION_BLOCK

// ---- POUs/HTTP/FB_TalkToGateway.TcPOU
FUNCTION_BLOCK FB_TalkToGateway
VAR_INPUT
    strIPAddress        : STRING;
    nPortNumber         : UINT;
    strDeviceID         : ARRAY[1..GVL_Const.cMaxVibrationDevices] OF STRING;
    bStopConnection     : BOOL;
    bResetError         : BOOL;
    bSendRequest        : BOOL; // NOT IMPLEMENTED YET
    eRequestType        : E_RequestType; // NOT IMPLEMENTED YET
    iRequestDeviceIndex : UINT; // NOT IMPLEMENTED YET
    tPollTime           : TIME;
END_VAR

VAR_OUTPUT
    bError           : BOOL;
    fbErrHist        : FB_HRErrHist; // error monitoring	
    aDeviceResponse  : ARRAY[1..GVL_Const.cMaxVibrationDevices] OF ST_ReceivedData; // data from device  // TODO write into
    strRequestOutput : STRING; // NOT IMPLEMENTED YET
	bProcessingRequest : BOOL;

END_VAR

VAR
    fbHttpClient : FB_IotHttpClient := (bKeepAlive         := TRUE,
                                        tConnectionTimeout := T#10S);
    fbGetDataFromHTTPAddr : GetDataFromSensorWorksHTTP;
    PollTimer             : TON;
    bGetData              : BOOL;
    i                     : UINT;
    nNumDevices           : UINT;
    bExecuteSend          : BOOL;
    strRequest            : STRING;
    buffstrRequest        : STRING;
    fbGateWayRequest      : FB_RequestToGateway;

END_VAR

VAR   // Qin
    bLogOnce : BOOL := TRUE;  // to make sure logging happens only once per cycle
END_VAR

IF bSendRequest THEN
    fbGateWayRequest(
        bExecute            := TRUE,
        eRequestType        := eRequestType,
        strIPAddress        := strIPAddress,
        nPortNumber         := nPortNumber,
        //iRequestDeviceIndex := iRequestDeviceIndex,
		iRequestDeviceIndex := 1,
        strDeviceID         := strDeviceID,
        fbClient            := fbHttpClient
    );
END_IF;


(**** ERROR HANDLING - NOT COMPLETED, NO RESET IMPLEMENTED YET ****)

IF strIPAddress = '' THEN
    fbErrHist.AddError(bErr := TRUE, hrErrCode := e_NoIPAddress, sErrSource := 'IP Address');
    bError := TRUE;
END_IF


IF nPortNumber = 0 THEN
    fbErrHist.AddError(bErr := TRUE, hrErrCode := e_NoPortNumber, sErrSource := 'Port Number');
    bError := TRUE;
END_IF

// Update connection details on disconnection
IF NOT fbHttpClient.bConfigured THEN
    fbHttpClient.sHostName := strIPAddress;
    fbHttpClient.nHostPort := nPortNumber;
    PollTimer.PT           := tPollTime;
END_IF

IF PollTimer.Q THEN // Normal data aqcuisition 
    bGetData := TRUE;
    i        := 1;
END_IF

IF bGetData THEN
    IF i > GVL_Const.cMaxVibrationDevices THEN
        bGetData := FALSE;
    ELSE

        IF strDeviceID[i] <> '' AND NOT fbGetDataFromHTTPAddr.bBusy THEN
            buffstrRequest := CONCAT('/device/', strDeviceID[i]);
            strRequest     := CONCAT(buffstrRequest, '/cache/latest');   // Builds up request to ask for data  replace with parameter/

            bExecuteSend := TRUE;
        ELSIF strDeviceID[i] = '' AND NOT fbGetDataFromHTTPAddr.bBusy THEN
            i            := i + 1; // Look for next array point
            strRequest   := '';    // clear
            bExecuteSend := FALSE;
        END_IF

        fbGetDataFromHTTPAddr(bSend := bExecuteSend, fbClient := fbHttpClient, strRequest := strRequest); // Function block to call the request for data

        IF fbGetDataFromHTTPAddr.bBusy AND bExecuteSend THEN
            bExecuteSend := FALSE; //reset trigger for next cycle, input above requires rising edge	
        END_IF

        IF NOT fbGetDataFromHTTPAddr.bBusy AND NOT fbGetDataFromHTTPAddr.bError AND strDeviceID[i] <> '' THEN
            aDeviceResponse[i] := fbGetDataFromHTTPAddr.jsonObatinedData;
            i                  := i + 1; // Look for next array point
        END_IF
    END_IF
END_IF

(****** Not finished, do not use ******
IF fbHttpClient.bConfigured AND bSendRequest AND NOT fbGateWayRequest.bBusy THEN
    fbGateWayRequest.bExecute            := TRUE;
    fbGateWayRequest.eRequestType        := eRequestType;
    fbGateWayRequest.strIPAddress        := strIPAddress;
    fbGateWayRequest.nPortNumber         := nPortNumber;
    fbGateWayRequest.iRequestDeviceIndex := iRequestDeviceIndex;
    fbGateWayRequest.strDeviceID         := strDeviceID;
ELSIF fbHttpClient.bConfigured AND bSendRequest AND fbGateWayRequest.bBusy THEN
    fbGateWayRequest.bExecute := FALSE;

END_IF

****** END OF COMMENT *****)

IF bStopConnection AND fbHttpClient.bConfigured THEN
    fbHttpClient.Disconnect();
ELSE
    fbHttpClient.Execute();
END_IF

PollTimer(IN := fbHttpClient.bConfigured AND NOT PollTimer.Q);

fbGateWayRequest(fbClient := fbHttpClient);

END_FUNCTION_BLOCK

// ---- POUs/HTTP/GetDataFromSensorWorksHTTP.TcPOU
FUNCTION_BLOCK GetDataFromSensorWorksHTTP
VAR_INPUT
    bSend       : BOOL;
    strRequest  : STRING; // := '/device/d5:d0:f9:30:83:d7/cache/latest'; // EXAMPLE REQUEST STRING
    bErrorReset : BOOL;
END_VAR
VAR_IN_OUT
    fbClient : FB_IotHttpClient;
END_VAR
VAR_OUTPUT
    bBusy            : BOOL;
    bError           : BOOL;
    jsonObatinedData : ST_ReceivedData;

END_VAR
VAR
    fbRequest  : FB_IotHttpRequest;
    fbJson     : FB_JsonDomParser;
    nState     : UDINT;
    RisingEdge : R_TRIG;

    bGetContentResult : BOOL;

    jsonDoc        : SJsonValue;
    jsonVal        : SJsonValue;
    sResultValue   : STRING;

    nReqCount      : UDINT;
    nResCount      : UDINT;
    nValidResCount : UDINT;
    nErrCount      : UDINT;
    sContent       : STRING(16000);

    jsonProp : SJsonValue;

    jsonDoc2        : SJsonValue;
    jsonIterator    : SJsonIterator;
    jsonIteratorEnd : SJsonIterator;
    i               : INT;
END_VAR

RisingEdge(CLK := bSend);

CASE nState OF
    0:
        IF RisingEdge.Q AND NOT bError THEN
			MEMSET(ADR(jsonObatinedData),0, SIZEOF(jsonObatinedData));
            IF fbRequest.SendRequest(sUri         := strRequest,
                                     fbClient     := fbClient,
                                     eRequestType := ETcIotHttpRequestType.HTTP_Get,
                                     0,
                                     0,
                                     0) THEN
                nState    := 1;
                nReqCount := nReqCount + 1;
                bBusy     := TRUE;
                bError    := FALSE;
            END_IF
        END_IF

        IF bErrorReset THEN
            nErrCount := 0;
            nReqCount := 0;
            nResCount := 0;
            bError    := FALSE;
        END_IF

    1:
        IF NOT fbRequest.bBusy THEN
            bError := TRUE;

            IF NOT fbRequest.bError THEN
                bGetContentResult := fbRequest.GetContent(pContent            := ADR(sContent),
                                                          nContentSize        := SIZEOF(sContent),
                                                          bSetNullTermination := TRUE);

                IF fbRequest.nStatusCode >= 200 AND fbRequest.nStatusCode < 300 THEN
                    jsonDoc := fbRequest.GetJsonDomContent(fbJson);

                    IF jsonDoc <> 0 THEN
                        nState         := 2;
                        nValidResCount := nValidResCount + 1;
                        bError         := FALSE;
                    END_IF

                    nResCount := nResCount + 1;
                END_IF
            END_IF

            IF bError THEN
                nErrCount := nErrCount + 1;
                bBusy     := FALSE;
                nState    := 0;
            END_IF
        END_IF

    2:

        jsonDoc2 := fbJson.ParseDocument(sContent);

        jsonProp := fbJson.FindMember(jsonDoc, 'uuid');

        IF (jsonProp <> 0) THEN
            jsonObatinedData.uuid := fbJson.GetString(jsonProp);
        END_IF

        jsonProp := fbJson.FindMember(jsonDoc, 'blename');

        IF (jsonProp <> 0) THEN
            jsonObatinedData.blename := fbJson.GetString(jsonProp);
        END_IF

        jsonProp := fbJson.FindMember(jsonDoc, 'name');

        IF (jsonProp <> 0) THEN
            jsonObatinedData.name := fbJson.GetString(jsonProp);
        END_IF

        jsonProp := fbJson.FindMember(jsonDoc, 'id');

        IF (jsonProp <> 0) THEN
            jsonObatinedData.id := fbJson.GetString(jsonProp);
        END_IF

        jsonProp := fbJson.FindMember(jsonDoc, 'time');

        IF (jsonProp <> 0) THEN
            jsonObatinedData.timestamp := fbJson.GetString(jsonProp);
        END_IF

        jsonProp := fbJson.FindMember(jsonDoc, 'rate');

        IF (jsonProp <> 0) THEN
            jsonObatinedData.rate := fbJson.GetInt(jsonProp);
        END_IF

        jsonProp := fbJson.FindMember(jsonDoc, 'trace');

        IF (jsonProp <> 0) THEN
            jsonObatinedData.trace := fbJson.GetInt(jsonProp);
        END_IF

        jsonProp := fbJson.FindMember(jsonDoc, 'count');

        IF (jsonProp <> 0) THEN
            jsonObatinedData.count := fbJson.GetInt(jsonProp);
        END_IF

        jsonProp := fbJson.FindMember(jsonDoc, 'gain');

        IF (jsonProp <> 0) THEN
            jsonObatinedData.gain := fbJson.GetInt(jsonProp);
        END_IF

        jsonProp := fbJson.FindMember(jsonDoc, 'calibration');

        IF (jsonProp <> 0) THEN
            jsonObatinedData.calibration := fbJson.GetDouble(jsonProp);
        END_IF

        jsonProp := fbJson.FindMember(jsonDoc, 'calibration_y');

        IF (jsonProp <> 0) THEN
            jsonObatinedData.calibration_y := fbJson.GetDouble(jsonProp);
        END_IF

        jsonProp := fbJson.FindMember(jsonDoc, 'calibration_z');

        IF (jsonProp <> 0) THEN
            jsonObatinedData.calibration_z := fbJson.GetDouble(jsonProp);
        END_IF

        jsonProp := fbJson.FindMember(jsonDoc, 'temperature');

        IF (jsonProp <> 0) THEN
            jsonObatinedData.temperature := fbJson.GetDouble(jsonProp);
        END_IF

        jsonProp := fbJson.FindMember(jsonDoc, 'battery');

        IF (jsonProp <> 0) THEN
            jsonObatinedData.battery := fbJson.GetDouble(jsonProp);
        END_IF

        jsonProp := fbJson.FindMember(jsonDoc, 'axes');

        IF (jsonProp <> 0) THEN
            jsonObatinedData.axes := fbJson.GetDouble(jsonProp);
        END_IF

        jsonProp := fbJson.FindMember(jsonDoc, 'mux_axis');

        IF (jsonProp <> 0) THEN
            jsonObatinedData.mux_axis := fbJson.GetDouble(jsonProp);
        END_IF

        jsonProp := fbJson.FindMember(jsonDoc, 'measure_rate');

        IF (jsonProp <> 0) THEN
            jsonObatinedData.measured_rate := fbJson.GetDouble(jsonProp);
        END_IF

        nState := 3;

    3:

        jsonProp := fbJson.FindMember(jsonDoc, 'value');

        IF (jsonProp <> 0) THEN
            jsonIterator    := fbJson.ArrayBegin(jsonProp);
            jsonIteratorEnd := fbJson.ArrayEnd(jsonProp);
            i               := 0;

            WHILE jsonIterator <> jsonIteratorEnd DO
                IF jsonProp <> 0 THEN
                    jsonObatinedData.value[i + 1] := fbJson.GetInt(jsonIterator);
                END_IF

                i            := i + 1;
                jsonIterator := fbJson.NextArray(jsonIterator);
            END_WHILE
        END_IF

        jsonProp := fbJson.FindMember(jsonDoc, 'value_y');

        IF (jsonProp <> 0) THEN
            jsonIterator    := fbJson.ArrayBegin(jsonProp);
            jsonIteratorEnd := fbJson.ArrayEnd(jsonProp);
            i               := 0;

            WHILE jsonIterator <> jsonIteratorEnd DO
                IF jsonProp <> 0 THEN
                    jsonObatinedData.value_y[i + 1] := fbJson.GetInt(jsonIterator);
                END_IF

                i            := i + 1;
                jsonIterator := fbJson.NextArray(jsonIterator);
            END_WHILE
        END_IF

        jsonProp := fbJson.FindMember(jsonDoc, 'value_z');

        IF (jsonProp <> 0) THEN
            jsonIterator    := fbJson.ArrayBegin(jsonProp);
            jsonIteratorEnd := fbJson.ArrayEnd(jsonProp);
            i               := 0;

            WHILE jsonIterator <> jsonIteratorEnd DO
                IF jsonProp <> 0 THEN
                    jsonObatinedData.value_z[i + 1] := fbJson.GetInt(jsonIterator);
                END_IF

                i            := i + 1;
                jsonIterator := fbJson.NextArray(jsonIterator);
            END_WHILE
        END_IF

        bBusy  := FALSE;
        nState := 0;

END_CASE

END_FUNCTION_BLOCK

// ---- POUs/HTTP/FB_RequestToGateway.TcPOU
FUNCTION_BLOCK FB_RequestToGateway
VAR_INPUT
    bExecute            : BOOL;
    eRequestType        : E_RequestType;
    strIPAddress        : STRING;
    nPortNumber         : UINT;
    iRequestDeviceIndex : UINT;
    strDeviceID         : ARRAY[1..GVL_Const.cMaxVibrationDevices] OF STRING;

END_VAR
VAR_IN_OUT
    fbClient : FB_IotHttpClient;
END_VAR
VAR_OUTPUT
    bDone      : BOOL;
    bBusy      : BOOL;
    bError     : BOOL;
    eErrorCode : E_TalkToGateway_Err;
    sContent   : STRING(80);   // not to get data
	//sContent   : ARRAY [0..16000] OF BYTE;  // Changed from STRING(8191)    // Qin
	//sContent : ARRAY [0..20] OF STRING(8000);  // 3 strings of 8000 chars each  Qin
	


END_VAR
VAR
    fbRequest : FB_IotHttpRequest;
    fbJson    : FB_JsonDomParser;

    nReqCount  : UDINT;
    strRequest : STRING;

    step              : E_RequestType;
    buffstrRequest    : STRING;
    bGetContentResult : BOOL;
    jsonDoc           : SJsonValue;
    nResCount         : UDINT;
    nValidResCount    : UDINT;
    nErrCount         : UDINT;

	strRequestOutput: STRING(255);
	
		// Debug variables   QIn
    nLen0 : INT;
    nLen1 : INT;
    nLen2 : INT;
    sFirst10_0 : STRING(10);
    sFirst10_1 : STRING(10);
    sFirst10_2 : STRING(10);
	sTail100: STRING(50);

	nLenContent: UDINT;
	nStartPos: UDINT;
	sContentTail: STRING(50);
	i: UDINT;
END_VAR

CASE step OF
    eIdle:

        IF bExecute THEN
			bError := FALSE;   // Qin
   		    eErrorCode := 0; // Reset error state
			//strRequestOutput := CONCAT('IP: ', CONCAT(strIPAddress, CONCAT(' / Error: ', INT_TO_STRING(eErrorCode))));   // for bebug

		
            IF (iRequestDeviceIndex < 1) OR (iRequestDeviceIndex > GVL_Const.cMaxVibrationDevices) THEN
                eErrorCode := e_DeviceIDOutsideLimits;
                step       := eERROR;
            ELSIF strDeviceID[iRequestDeviceIndex] = '' THEN
                eErrorCode := e_DeviceIDNotFound;
                step       := eERROR;
            ELSE

                step := eRequestType;
            END_IF
        END_IF

    (**** This could be implemented in various ways ****)
    (**** depending on what you prefer, here are some quick examples ****)

    eSampleRate:
        buffstrRequest := CONCAT('/device/', strDeviceID[iRequestDeviceIndex]);
        strRequest     := CONCAT(buffstrRequest, '/parameter/sample_rate');
        step           := eRequestSend;

    eTraceLen:
        buffstrRequest := CONCAT('/device/', strDeviceID[iRequestDeviceIndex]);
        strRequest     := CONCAT(buffstrRequest, '/parameter/tracelen');
        step           := eRequestSend;

    eMode:
        buffstrRequest := CONCAT('/device/', strDeviceID[iRequestDeviceIndex]);
        strRequest     := CONCAT(buffstrRequest, '/parameter/mode');
        step           := eRequestSend;
	
	eViewRequest:   // Qin
		buffstrRequest := CONCAT('/device/', strDeviceID[iRequestDeviceIndex]);
		strRequest     := CONCAT(buffstrRequest, '/cache/latest');
		
        step           := eRequestSend;

    (********* End of string building *********)
    eRequestSend:
        IF fbRequest.SendRequest(sUri         := strRequest,
                                 fbClient     := fbClient,
                                 eRequestType := ETcIotHttpRequestType.HTTP_Get,
                                 0,
                                 0,
                                 0) THEN
            step      := eGetData;
            nReqCount := nReqCount + 1;
            bBusy     := TRUE;
            bError    := FALSE;
        END_IF

    eGetData:
        IF NOT fbRequest.bBusy THEN
            bError := TRUE;

            IF NOT fbRequest.bError THEN
                bGetContentResult := fbRequest.GetContent(pContent            := ADR(sContent),
                                                          nContentSize        := SIZEOF(sContent),
                                                          bSetNullTermination := TRUE);

                IF fbRequest.nStatusCode >= 200 AND fbRequest.nStatusCode < 300 THEN
                    jsonDoc := fbRequest.GetJsonDomContent(fbJson);

                    IF jsonDoc <> 0 THEN
                        (**** Process data for which member is desired ****)
                        step := eProcess;
                        (********)
                        nValidResCount := nValidResCount + 1;
                        bError         := FALSE;
                    END_IF

                    nResCount := nResCount + 1;
                END_IF
            END_IF

            IF bError THEN
                nErrCount  := nErrCount + 1;
                bBusy      := FALSE;
                eErrorCode := e_JSONRequestError;
                step       := eERROR;
            END_IF
        END_IF

    eProcess:
        bBusy := FALSE;
        step  := eIdle;

    eERROR:
// Error handling

END_CASE

// Qin debug sContent
nLenContent := LEN2(ADR(sContent)); // Correct usage with ADR
IF nLenContent > 50 THEN
    nStartPos := nLenContent - 50 + 1; // Position for last 100 chars
ELSE
    nStartPos := 1; // If string shorter than 100, start at beginning
END_IF;
//sContentTail := MID2(ADR(sContent), nStartPos, 100); // Extract substring// MID2 not available
FOR i := 0 TO 49 DO
    sContentTail[i] := sContent[nStartPos + i - 1];
END_FOR

END_FUNCTION_BLOCK

// ---- POUs/CM_Collection/CM_Sim.TcPOU
PROGRAM CM_Sim
VAR CONSTANT
		    cInitSource			: ST_MA_MultiArray_InitPars 
							:= ( eTypeCode := eMA_TypeCode_LREAL, nDims := 2, aDimSizes := [ GVL_Const.cChannels, GVL_Const.cBufferLength]);

END_VAR
VAR
		(* Input from aBuffer to fbSource *)
	fbSource_ISO			: FB_CMA_Source :=(	stInitPars := cInitSource, 
											nOwnID := eID_SimSource, 
											aDestIDs := [eID_SimISO],
											nResultBuffers := 4);		// Initialize source buffers
	
	fbSink				: FB_CMA_Sink := (nOwnID := eID_SimSinkISO);

	fbErrHist			: FB_HRErrHist; // error monitoring	

	
	(* Classify calculated RMS values *)
	nCountResults		  : ULINT;	
	bCalculate			  : BOOL;
	nChannel              : UDINT;
	ISOClassIs_Vel        : ARRAY[1..GVL_Const.cChannels] OF E_IsoClass;
	ISOClassIs_Displ      : ARRAY[1..GVL_Const.cChannels] OF E_IsoClass;	
	
	(* Buffer variables for calculation *)
	Ch1VelRMS : LREAL;
	Ch1DisplRMS : LREAL;
	Ch2VelRMS : LREAL;
	Ch2DisplRMS : LREAL;
	
	(* output *)
	ISO_10816_Classification AT%Q* : E_IsoClass;
	
	intMachineSelected: USINT := 1;
	intElasticitySelected: USINT :=1;
	
	Ch1AccRMS: LREAL;
	Ch2AccRMS: LREAL;
END_VAR
VAR CONSTANT
	MachineDisplISOClassLimit: E_IsoClass := 3;
	MachineVelISOClassLimit: E_IsoClass := 3;
END_VAR

(* Collect raw data and send it for calculation *)
SourceData();

(* Get results from RMS *)
SinkData();

(* Classify the data *)
Classification();

ACTION Classification:
// define class according to ISO 10816-3 based on velocity and displacement data for each measurement channel
IF bCalculate THEN
	Ch1AccRMS := GLOBAL.aSimRMSResult[1][1];
	Ch1VelRMS := GLOBAL.aSimRMSResult[1][2];
	Ch1DisplRMS := GLOBAL.aSimRMSResult[1][3];
	Ch2AccRMS := GLOBAL.aSimRMSResult[2][1];
	Ch2VelRMS := GLOBAL.aSimRMSResult[2][2];
	Ch2DisplRMS := GLOBAL.aSimRMSResult[2][3];	
	
	IF NOT lrealisnan(Ch1VelRMS) THEN 

		nCountResults := fbSink.nCntResults;
		
		// do for each channel
		FOR nChannel := 1 TO GVL_Const.cChannels DO
			
			// evaluate velocity data
			ISOClassIs_Vel[nChannel] := E_IsoClass.A;
			IF GLOBAL.aSimRMSResult[nChannel][2] > GVL_Const.cISOClassDef_Velocity[intMachineSelected,intElasticitySelected,3] THEN
				ISOClassIs_Vel[nChannel] := E_IsoClass.D;
			ELSIF GLOBAL.aSimRMSResult[nChannel][2] > GVL_Const.cISOClassDef_Velocity[intMachineSelected,intElasticitySelected,2] THEN
				ISOClassIs_Vel[nChannel] := E_IsoClass.C;
			ELSIF GLOBAL.aSimRMSResult[nChannel][2] > GVL_Const.cISOClassDef_Velocity[intMachineSelected,intElasticitySelected,1] THEN
				ISOClassIs_Vel[nChannel] := E_IsoClass.B;
			END_IF;  
			
			// evaluate displacement data
			ISOClassIs_Displ[nChannel] := E_IsoClass.A;
			IF GLOBAL.aSimRMSResult[nChannel][3] > GVL_Const.cISOClassDef_Displ[intMachineSelected,intElasticitySelected,3] THEN
				ISOClassIs_Displ[nChannel] := E_IsoClass.D;
			ELSIF GLOBAL.aSimRMSResult[nChannel][3] > GVL_Const.cISOClassDef_Displ[intMachineSelected,intElasticitySelected,2] THEN
				ISOClassIs_Displ[nChannel] := E_IsoClass.C;
			ELSIF GLOBAL.aSimRMSResult[nChannel][3] > GVL_Const.cISOClassDef_Displ[intMachineSelected,intElasticitySelected,1] THEN
				ISOClassIs_Displ[nChannel] := E_IsoClass.B;
			END_IF;	
									
		END_FOR;
		
		// according to ISO 10816-3 select worst case 		
		ISO_10816_Classification := E_IsoClass.A;
		FOR  nChannel := 1 TO GVL_Const.cChannels DO 
			IF ISOClassIs_Vel[nChannel] >  ISO_10816_Classification THEN
				ISO_10816_Classification := ISOClassIs_Vel[nChannel];
			END_IF
			IF ISOClassIs_Displ[nChannel] >  ISO_10816_Classification THEN
				ISO_10816_Classification := ISOClassIs_Displ[nChannel];
			END_IF
		END_FOR;
		
		

		
	ELSE
		// result is NaN... code here what to do. 
		
	END_IF;
	
END_IF
END_ACTION

ACTION SinkData:
(* Push results to sink *)
fbSink.Output2D(	pDataOut 		:= ADR(GLOBAL.aSimRMSResult), 
					nDataOutSize 	:= SIZEOF(GLOBAL.aSimRMSResult), 
					eElementType 	:= eMA_TypeCode_LREAL, 
					nWorkDim0 		:= 0,
					nWorkDim1 		:= 1,
					nElementsDim0	:= 0,
					nElementsDim1	:= 0,
					pStartIndex 	:= 0,
					nOptionPars		:= 0,
					bNewResult		=> bCalculate );
					
IF fbSink.bError THEN
	fbErrHist.AddError(bErr:=TRUE, hrErrCode:=fbSink.hrErrorCode, sErrSource:='CM_Sim.fbSink'); // error monitoring
	// ToDo: if error
END_IF
END_ACTION

ACTION SourceData:
// Collection
fbSource_ISO.Input2D(pDataIn 			:= ADR(GLOBAL.aSimBuffer),
				  nDataInSize 		:= SIZEOF(GLOBAL.aSimBuffer), 
				  eElementType 		:= eMA_TypeCode_LREAL,
				  nWorkDim0			:= 0,
				  nWorkDim1			:= 1,
				  pStartIndex		:= 0,
				  nOptionPars		:= 0 ); 
				  
// Check for errors
IF fbSource_ISO.bError THEN
	fbErrHist.AddError(bErr:=TRUE, hrErrCode:=fbSource_ISO.hrErrorCode, sErrSource:='CM_Sim.SourceData.fbSource_ISO');	
END_IF
END_ACTION

END_PROGRAM

// ---- POUs/CM_Collection/CM_SensorWorks_Sensor1.TcPOU
PROGRAM CM_SensorWorks_Sensor1
VAR CONSTANT
		    cInitSource			: ST_MA_MultiArray_InitPars 
							:= ( eTypeCode := eMA_TypeCode_LREAL, nDims := 2, aDimSizes := [GVL_Const.cSensorSampleChannels,GVL_Const.cSensorPacket]);

END_VAR
VAR
		(* Input from aSimBuffer to fbSource *)
	fbSource_SensorWorks			: FB_CMA_Source :=(	stInitPars := cInitSource, 
											nOwnID := eID_SW_Source_Device_1, 
											aDestIDs := [eID_SW_ISO_Device_1],
											nResultBuffers := 4);		// Initialize source buffers

											//aDestIDs := [eID_SensorWorksISO,eID_SensorWorksSpectrum]);
	
	fbSinkISO						: FB_CMA_Sink := (nOwnID := eID_SW_Sink_Device_1);
//	fbSinkMagSpec					: FB_CMA_Sink := (nOwnID := eID_SensorWorkSinkSpectrum);

	fbErrHist						: FB_HRErrHist; // error monitoring	

	(* Calculate triggers *)
	bCalculateISO					: BOOL;
	
	(* Buffer variables for calculation *)
	Ch1VelRMS 						: LREAL;
	Ch1DisplRMS 					: LREAL;
	Ch1AccRMS: LREAL;

	Ch2VelRMS 						: LREAL;
	Ch2DisplRMS 					: LREAL;
	Ch2AccRMS: LREAL;

	(* output *)
	ISO_10816_Classification AT%Q* : E_IsoClass;
	
	intMachineSelected: USINT := 1;
	intElasticitySelected: USINT :=1;
	
	(* Classify calculated RMS values *)
	nCountResults		  : ULINT;	
	bCalculate			  : BOOL;
	nChannel              : UDINT;
	ISOClassIs_Vel        : E_IsoClass;
	ISOClassIs_Displ      : E_IsoClass;	

	bNewSensorDataAvailable: BOOL := TRUE;
	i: UDINT;
	testwave: FB_FunctionGenerator_1;
	testfq: LREAL := 400;
	fSetAmplitude1: LREAL := 10;
	strOldTS: STRING;
END_VAR

VAR CONSTANT
	MachineDisplISOClassLimit: E_IsoClass := 3;
	MachineVelISOClassLimit: E_IsoClass := 3;
END_VAR

(* Collect raw data and send it for calculation *)
SourceData();

(* Get results from RMS *)
SinkData();

(* Classify the data *)
Classification();

ACTION Classification:
// define class according to ISO 10816-3 based on velocity and displacement data for each measurement channel
IF bCalculateISO THEN
	Ch1AccRMS := GLOBAL.aSensorWorkISOHTTPResult[1][1];
	Ch1VelRMS := GLOBAL.aSensorWorkISOHTTPResult[1][2];
	Ch1DisplRMS := GLOBAL.aSensorWorkISOHTTPResult[1][3];

	
	IF NOT lrealisnan(Ch1VelRMS) THEN 

		nCountResults := fbSinkISO.nCntResults;
		

			
			// evaluate velocity data
			ISOClassIs_Vel := E_IsoClass.A;
			IF GLOBAL.aSensorWorkISOHTTPResult[1][2] > GVL_Const.cISOClassDef_Velocity[intMachineSelected,intElasticitySelected,3] THEN
				ISOClassIs_Vel := E_IsoClass.D;
			ELSIF GLOBAL.aSensorWorkISOHTTPResult[1][2] > GVL_Const.cISOClassDef_Velocity[intMachineSelected,intElasticitySelected,2] THEN
				ISOClassIs_Vel := E_IsoClass.C;
			ELSIF GLOBAL.aSensorWorkISOHTTPResult[1][2] > GVL_Const.cISOClassDef_Velocity[intMachineSelected,intElasticitySelected,1] THEN
				ISOClassIs_Vel := E_IsoClass.B;
			END_IF;  
			
			// evaluate displacement data
			ISOClassIs_Displ := E_IsoClass.A;
			IF GLOBAL.aSensorWorkISOHTTPResult[1][3] > GVL_Const.cISOClassDef_Displ[intMachineSelected,intElasticitySelected,3] THEN
				ISOClassIs_Displ := E_IsoClass.D;
			ELSIF GLOBAL.aSensorWorkISOHTTPResult[1][3] > GVL_Const.cISOClassDef_Displ[intMachineSelected,intElasticitySelected,2] THEN
				ISOClassIs_Displ := E_IsoClass.C;
			ELSIF GLOBAL.aSensorWorkISOHTTPResult[1][3] > GVL_Const.cISOClassDef_Displ[intMachineSelected,intElasticitySelected,1] THEN
				ISOClassIs_Displ := E_IsoClass.B;
			END_IF;	
									
		
		// according to ISO 10816-3 select worst case 		
		ISO_10816_Classification := E_IsoClass.A;
			IF ISOClassIs_Vel >  ISO_10816_Classification THEN
				ISO_10816_Classification := ISOClassIs_Vel;
			END_IF
			IF ISOClassIs_Displ >  ISO_10816_Classification THEN
				ISO_10816_Classification := ISOClassIs_Displ;
			END_IF

		
	ELSE
		// result is NaN... code here what to do. 
		
	END_IF;
	
END_IF
END_ACTION

ACTION SinkData:
(* Push results to sink *)
fbSinkISO.Output2DStd(	pDataOut 		:= ADR(GLOBAL.aSensorWorkISOHTTPResult[1]), 
					nDataOutSize 	:= SIZEOF(GLOBAL.aSensorWorkISOHTTPResult[1]), 
					eElementType 	:= eMA_TypeCode_LREAL, 
					nOptionPars		:= 0,
					
					bNewResult		=> bCalculateISO );
					
IF fbSinkISO.bError THEN
	fbErrHist.AddError(bErr:=TRUE, hrErrCode:=fbSinkISO.hrErrorCode, sErrSource:='CM_SensorWorks_Sensor1.fbSinkISO'); // error monitoring
	// ToDo: if error
END_IF
END_ACTION

ACTION SourceData:

IF GLOBAL.stSensorWorksHTTPSensorData[1].timestamp <> strOldTS THEN
    FOR i := 1 TO GVL_Const.cSensorPacket DO
        GLOBAL.aSensorWorksHTTPInput[1][i] := GLOBAL.stSensorWorksHTTPSensorData[1].value[i] * GLOBAL.stSensorWorksHTTPSensorData[1].calibration;
    END_FOR

    bNewSensorDataAvailable := TRUE;
END_IF

// TODO value follow timestamp



// Collection
IF bNewSensorDataAvailable THEN
    // Check to make sure code works
    (*	
	testwave(
	
			bEnable:= TRUE, 
			fFrequency 	:= testfq,
			fAmplitude 	:= 100,
			eFunction 	:= E_FunctionType.Sine,
			aSignal		:= GLOBAL.aSensorWorksHTTPInput[1]);	
	// end of signal generation
*)

    fbSource_SensorWorks.Input2DStd(pDataIn      := ADR(GLOBAL.aSensorWorksHTTPInput[1]),
                                    nDataInSize  := SIZEOF(GLOBAL.aSensorWorksHTTPInput[1]),
                                    eElementType := eMA_TypeCode_LREAL,
                                    nOptionPars  := Tc3_CM.cCMA_Option_MarkInterruption);

    bNewSensorDataAvailable := FALSE; // reset flag
    //testwave.bEnable := FALSE;
END_IF

// Check for errors
IF fbSource_SensorWorks.bError THEN
    fbErrHist.AddError(bErr := TRUE, hrErrCode := fbSource_SensorWorks.hrErrorCode, sErrSource := 'CM_SensorWorks_Sensor1.SourceData');
END_IF

strOldTS := GLOBAL.stSensorWorksHTTPSensorData[1].timestamp;
END_ACTION

END_PROGRAM

// ---- FUBs/FB_FunctionGenerator_1.TcPOU
// generates a signal build up by the specified function type. v1.6
FUNCTION_BLOCK FB_FunctionGenerator_1
VAR_INPUT
	bEnable		: BOOL 	:= TRUE;	// set TRUE to generate the specified signal; set FALSE to reset the signal buffer
	fFrequency	: LREAL := 1000;	// in [Hz]
	fAmplitude	: LREAL := 1;
	fOffset		: LREAL	:= 0;	
	nDutyCycle	: UINT 	:= 50;		// in [%] (for pulse function)
	eFunction	: E_FunctionType := E_FunctionType.Sine;	
END_VAR
VAR_IN_OUT
	aSignal		: ARRAY[1..GVL_Const.cSensorPacket] OF LREAL;
END_VAR
VAR_OUTPUT
	bError		: BOOL;
END_VAR

VAR
	bInit						: BOOL := TRUE;
	fbGetTaskIdx				: GETCURTASKINDEX;
	
	fLastFrequency				: LREAL;		// in [Hz]
	fLastAmplitude				: LREAL;
	fLastOffset					: LREAL;
	nLastDutyCycle				: UINT;
	eLastFunction				: E_FunctionType;
	
	nSamples					: UDINT;
	fCycleTime					: LREAL;		// in [s]
	fDelta						: LREAL;		// amplitude delta per sample
	fPhase						: LREAL;		// in [°]
	nSign						: INT := 1;		// 1 or -1
	fLastSignalValue			: LREAL;		// amplitude
	fPeriod						: LREAL;		// in [s]
	fAngularIncrement			: LREAL;		// in [°]
	fAngularIncrementPerCycle	: LREAL;		// in [°]
	fAngularIncrementPerSample	: LREAL;		// in [°]
	(* for modulated signal (carrier signal without offset) *)
	fCarrierFrequency					: LREAL := 500;	// in [Hz] (sine)
	fCarrierAmplitude					: LREAL := 1;
	fCarrierPeriod						: LREAL;		// in [s]
	fCarrierAngularIncrement			: LREAL;		// in [°]
	fCarrierAngularIncrementPerCycle	: LREAL;		// in [°]
	fCarrierAngularIncrementPerSample	: LREAL;		// in [°]
				
END_VAR

IF bEnable THEN
	IF fLastFrequency <> fFrequency THEN
		bInit := TRUE; // For automatic initializing
		fLastFrequency := fFrequency;
	END_IF
	IF fLastAmplitude <> fAmplitude THEN
		bInit := TRUE; // For automatic initializing
		fLastAmplitude := fAmplitude;
	END_IF
	IF fLastOffset <> fOffset THEN
		bInit := TRUE; // For automatic initializing
		fLastOffset := fOffset;
	END_IF
	IF nLastDutyCycle <> nDutyCycle THEN
		bInit := TRUE; // For automatic initializing
		nLastDutyCycle := nDutyCycle;
	END_IF
	IF eLastFunction <> eFunction THEN
		bInit := TRUE; // For automatic initializing
		eLastFunction := eFunction;
	END_IF
	IF bInit THEN
		// Get task info	
		fbGetTaskIdx();
		fCycleTime := UDINT_TO_LREAL(TwinCAT_SystemInfoVarList._TaskInfo[fbGetTaskIdx.index].CycleTime) (*100ns*) / (10.0 * 1000.0 * 1000.0);	
		fLastSignalValue := 0;
		nSign := 1;
		fAngularIncrement := 0;
		// Flush out old data
		MEMSET(ADR(aSignal), 0, SIZEOF(aSignal));
		IF fFrequency > 0 AND fCycleTime > 0 THEN		
			// Calculate period, increments per plc cycle, increment per oversample
			IF GVL_Const.cSensorPacket > 0 THEN			
				IF eFunction = E_FunctionType.Sine THEN
					fPeriod := 1/fFrequency;
					fAngularIncrementPerCycle := 360*(fCycleTime/fPeriod);
					fAngularIncrementPerSample := fAngularIncrementPerCycle/GVL_Const.cSensorPacket;
					// no phase adjustment
					bInit := FALSE;	
				ELSIF eFunction = E_FunctionType.Square	THEN
					fPeriod := 1/fFrequency;
					fAngularIncrementPerCycle  := 360*(fCycleTime/fPeriod);
					fAngularIncrementPerSample := fAngularIncrementPerCycle/GVL_Const.cSensorPacket;
					fPhase := 0.5*360;
					bInit := FALSE;
				ELSIF eFunction = E_FunctionType.Pulse THEN
					fPeriod := 1/fFrequency;
					fAngularIncrementPerCycle  := 360*(fCycleTime/fPeriod);
					fAngularIncrementPerSample := fAngularIncrementPerCycle/GVL_Const.cSensorPacket;
					IF nDutyCycle > 100 THEN
						nDutyCycle := 100;
					END_IF
					fPhase := (UDINT_TO_LREAL(nDutyCycle)/100)*360;
					bInit := FALSE;					
				ELSIF eFunction = E_FunctionType.Triangular THEN
					fPeriod := 1/fFrequency;				
					fAngularIncrementPerCycle  := 360*(fCycleTime/fPeriod);
					fAngularIncrementPerSample := fAngularIncrementPerCycle/GVL_Const.cSensorPacket;
					fPhase := 0.5*360; 
					fDelta := 4*(fAmplitude/(360/fAngularIncrementPerSample));				
					bInit := FALSE;
				ELSIF eFunction = E_FunctionType.Sawtooth THEN
					fPeriod := 1/fFrequency;			
					fAngularIncrementPerCycle  := 360*(fCycleTime/fPeriod);		
					fAngularIncrementPerSample := fAngularIncrementPerCycle/GVL_Const.cSensorPacket;
					fDelta := fAmplitude/(360/fAngularIncrementPerSample);
					bInit := FALSE;
				ELSIF eFunction = E_FunctionType.AM THEN
					fPeriod := 1/fFrequency;
					fAngularIncrementPerCycle := 360*(fCycleTime/fPeriod);
					fAngularIncrementPerSample := fAngularIncrementPerCycle/GVL_Const.cSensorPacket;
					// no phase adjustment
					fCarrierPeriod := 1/fCarrierFrequency;
					fCarrierAngularIncrementPerCycle := 360*(fCycleTime/fCarrierPeriod);
					fCarrierAngularIncrementPerSample := fCarrierAngularIncrementPerCycle/GVL_Const.cSensorPacket;				
					// no phase adjustment	
					bInit := FALSE;
				ELSE
					bError := TRUE;	
				END_IF
			ELSE
				bError := TRUE;
			END_IF
		ELSE
			bError := TRUE;
		END_IF
	END_IF
	
	// Enable function generator
	IF NOT bError THEN		
		CASE eFunction OF		
			// sine: typical for vibrations originating from rotating machine
			E_FunctionType.Sine: Sine();
			
			// square: mixed sine signals good for analyzing spectrum				
			E_FunctionType.Square: Square();
			
			// pulse: mixed sine signals good for analyzing spectrum				
			E_FunctionType.Pulse: Pulse();
	
			// sawtooth: ramp-type vibrations, continuously increasing			
			E_FunctionType.Sawtooth: Sawtooth();
		
			// triangular: mixed sine signals good for analyzing spectrum
			E_FunctionType.Triangular: Triangular();
		
			// amplitude modulation: typical for vibrations originating from gear-tooth failure or bearing faults
			// Carrier signal with own frequency and amplitude		
			E_FunctionType.AM: AM();				
		END_CASE
	END_IF
ELSE
	// Flush out old data
	MEMSET(ADR(aSignal), 0, SIZEOF(aSignal));
	
	bInit := TRUE;
	bError := FALSE;
END_IF

METHOD PRIVATE AM
VAR_INPUT
END_VAR
{warning disable C0371}

FOR nSamples := 1 TO GVL_Const.cSensorPacket DO
	// base signal * carrier signal
	aSignal[nSamples] := ( fAmplitude*SIN(2*PI*(fAngularIncrement+(nSamples-1)*fAngularIncrementPerSample)/360) + fOffset )
							* ( fCarrierAmplitude*SIN(2*PI*(fCarrierAngularIncrement+(nSamples-1)*fCarrierAngularIncrementPerSample)/360) );
END_FOR
// Increment angular positions
fAngularIncrement := fAngularIncrement + fAngularIncrementPerCycle;
fCarrierAngularIncrement := fCarrierAngularIncrement + fCarrierAngularIncrementPerCycle;

{warning restore C0371}
END_METHOD

METHOD PRIVATE Pulse
VAR_INPUT
END_VAR
{warning disable C0371}

FOR nSamples := 1 TO GVL_Const.cSensorPacket DO
	// For pulse wave (unequal phases)
	IF (fAngularIncrement >= 360) THEN
		fAngularIncrement := fAngularIncrement - DINT_TO_LREAL(LREAL_TO_DINT(fAngularIncrement/360))*360;
		// or with Tc2_Math library: fAngularIncrement := LMOD(fAngularIncrement,360);
	END_IF
	IF (fAngularIncrement < fPhase) THEN
		nSign := 1;		
	ELSIF (fAngularIncrement >= fPhase) THEN
		nSign := 0;
	END_IF
	fAngularIncrement := fAngularIncrement + fAngularIncrementPerSample;
	
	aSignal[nSamples] := nSign*fAmplitude;
	
	aSignal[nSamples] := aSignal[nSamples] + fOffset;
END_FOR

{warning restore C0371}
END_METHOD

METHOD PRIVATE Sawtooth
VAR_INPUT
END_VAR
{warning disable C0371}

FOR nSamples := 1 TO GVL_Const.cSensorPacket DO
	// For sawtooth wave (equal phase = period/2)
	IF (fAngularIncrement >= 360) THEN
		fAngularIncrement := fAngularIncrement - DINT_TO_LREAL(LREAL_TO_DINT(fAngularIncrement/360))*360;
		// or with Tc2_Math library: fAngularIncrement := LMOD(fAngularIncrement,360);
		fLastSignalValue := fLastSignalValue -fAmplitude;
	END_IF
	fAngularIncrement := fAngularIncrement + fAngularIncrementPerSample;

	aSignal[nSamples] := fLastSignalValue + fDelta;

	// Store last sample
	fLastSignalValue := aSignal[nSamples];
	
	aSignal[nSamples] := aSignal[nSamples] + fOffset;					
END_FOR	

{warning restore C0371}
END_METHOD

METHOD PRIVATE Sine
VAR_INPUT
END_VAR
{warning disable C0371}

FOR nSamples := 1 TO GVL_Const.cSensorPacket DO
	aSignal[nSamples] := fAmplitude*SIN(2*PI*(fAngularIncrement+(nSamples-1)*fAngularIncrementPerSample)/360);

	aSignal[nSamples] := aSignal[nSamples] + fOffset;
END_FOR

// Increment angular position
fAngularIncrement := fAngularIncrement + fAngularIncrementPerCycle;

{warning restore C0371}
END_METHOD

METHOD PRIVATE Square
VAR_INPUT
END_VAR
{warning disable C0371}

FOR nSamples := 1 TO GVL_Const.cSensorPacket DO
	// For square wave (equal phase = period/2)
	IF (fAngularIncrement >= 360) THEN
		fAngularIncrement := fAngularIncrement - DINT_TO_LREAL(LREAL_TO_DINT(fAngularIncrement/360))*360;
		// or with Tc2_Math library: fAngularIncrement := LMOD(fAngularIncrement,360);
	END_IF
	IF (fAngularIncrement < fPhase) THEN
		nSign := 1;
	ELSIF (fAngularIncrement >= fPhase) THEN
		nSign := -1;
	END_IF
	fAngularIncrement := fAngularIncrement + fAngularIncrementPerSample;
	
	aSignal[nSamples] := nSign*fAmplitude;
	
	aSignal[nSamples] := aSignal[nSamples] + fOffset;
END_FOR

{warning restore C0371}
END_METHOD

METHOD PRIVATE Triangular
VAR_INPUT
END_VAR
{warning disable C0371}

FOR nSamples := 1 TO GVL_Const.cSensorPacket DO
	IF (fAngularIncrement >= 360) THEN
		fAngularIncrement := fAngularIncrement - DINT_TO_LREAL(LREAL_TO_DINT(fAngularIncrement/360))*360;
		// or with Tc2_Math library: fAngularIncrement := LMOD(fAngularIncrement,360);
	END_IF
	// Negative delta -> Positive delta
	IF fAngularIncrement < fPhase/2 THEN	
		nSign := 1;		
	ELSIF fAngularIncrement >= fPhase/2 AND fAngularIncrement < 3*fPhase/2 THEN
		nSign := -1;
	ELSIF fAngularIncrement >= 3*fPhase/2 THEN
		nSign := 1;	
	END_IF
	fAngularIncrement := fAngularIncrement + fAngularIncrementPerSample;
	
	aSignal[nSamples] := fLastSignalValue + nSign*fDelta;
	IF aSignal[nSamples] > fAmplitude THEN
		aSignal[nSamples] := aSignal[nSamples] - 2*(aSignal[nSamples]-fAmplitude);
	ELSIF aSignal[nSamples] < (-1)*fAmplitude THEN
		aSignal[nSamples] := aSignal[nSamples] - 2*(aSignal[nSamples]+fAmplitude);
	END_IF
	
	// Store last sample
	fLastSignalValue := aSignal[nSamples];		
	
	aSignal[nSamples] := aSignal[nSamples] + fOffset;
END_FOR

{warning restore C0371}
END_METHOD

END_FUNCTION_BLOCK

// ---- POUs/CM_Collection/CM_SensorWorks_Sensor2.TcPOU
PROGRAM CM_SensorWorks_Sensor2
VAR CONSTANT
		    cInitSource			: ST_MA_MultiArray_InitPars 
							:= ( eTypeCode := eMA_TypeCode_LREAL, nDims := 2, aDimSizes := [GVL_Const.cSensorSampleChannels,GVL_Const.cSensorPacket]);
END_VAR
VAR
		(* Input from aSimBuffer to fbSource *)
	fbSource_SensorWorks			: FB_CMA_Source :=(	stInitPars := cInitSource, 
											nOwnID := eID_SW_Source_Device_2, 
											aDestIDs := [eID_SW_ISO_Device_2],
											nResultBuffers := 4);		// Initialize source buffers

	
	fbSinkISO						: FB_CMA_Sink := (nOwnID := eID_SW_Sink_Device_2);
	fbErrHist						: FB_HRErrHist; // error monitoring	
	(* Calculate triggers *)
	bCalculateISO					: BOOL;
	(* Buffer variables for calculation *)
	Ch1VelRMS 						: LREAL;
	Ch1DisplRMS 					: LREAL;
	Ch1AccRMS: LREAL;

	Ch2VelRMS 						: LREAL;
	Ch2DisplRMS 					: LREAL;
	Ch2AccRMS: LREAL;

	(* output *)
	ISO_10816_Classification AT%Q* : E_IsoClass;
	
	intMachineSelected: USINT := 1;
	intElasticitySelected: USINT :=1;
	
	(* Classify calculated RMS values *)
	nCountResults		  : ULINT;	
	bCalculate			  : BOOL;
	nChannel              : UDINT;
	ISOClassIs_Vel        : E_IsoClass;
	ISOClassIs_Displ      : E_IsoClass;	

	bNewSensorDataAvailable: BOOL := TRUE;
	i: UDINT;
	testwave: FB_FunctionGenerator_1;
	testfq: LREAL := 400;
	fSetAmplitude1: LREAL := 10;
	strOldTS: STRING;
END_VAR

VAR CONSTANT
	MachineDisplISOClassLimit: E_IsoClass := 3;
	MachineVelISOClassLimit: E_IsoClass := 3;
END_VAR

(* Collect raw data and send it for calculation *)
SourceData();

(* Get results from RMS *)
SinkData();

(* Classify the data *)
Classification();

ACTION Classification:
// define class according to ISO 10816-3 based on velocity and displacement data for each measurement channel
IF bCalculateISO THEN
    Ch1AccRMS   := GLOBAL.aSensorWorkISOHTTPResult[2][1];
    Ch1VelRMS   := GLOBAL.aSensorWorkISOHTTPResult[2][2];
    Ch1DisplRMS := GLOBAL.aSensorWorkISOHTTPResult[2][3];

    IF NOT lrealisnan(Ch1VelRMS) THEN

        nCountResults := fbSinkISO.nCntResults;

        // evaluate velocity data
        ISOClassIs_Vel := E_IsoClass.A;
        IF GLOBAL.aSensorWorkISOHTTPResult[2][2] > GVL_Const.cISOClassDef_Velocity[intMachineSelected, intElasticitySelected, 3] THEN
            ISOClassIs_Vel := E_IsoClass.D;
        ELSIF GLOBAL.aSensorWorkISOHTTPResult[2][2] > GVL_Const.cISOClassDef_Velocity[intMachineSelected, intElasticitySelected, 2] THEN
            ISOClassIs_Vel := E_IsoClass.C;
        ELSIF GLOBAL.aSensorWorkISOHTTPResult[2][2] > GVL_Const.cISOClassDef_Velocity[intMachineSelected, intElasticitySelected, 1] THEN
            ISOClassIs_Vel := E_IsoClass.B;
        END_IF;

        // evaluate displacement data
        ISOClassIs_Displ := E_IsoClass.A;
        IF GLOBAL.aSensorWorkISOHTTPResult[2][3] > GVL_Const.cISOClassDef_Displ[intMachineSelected, intElasticitySelected, 3] THEN
            ISOClassIs_Displ := E_IsoClass.D;
        ELSIF GLOBAL.aSensorWorkISOHTTPResult[2][3] > GVL_Const.cISOClassDef_Displ[intMachineSelected, intElasticitySelected, 2] THEN
            ISOClassIs_Displ := E_IsoClass.C;
        ELSIF GLOBAL.aSensorWorkISOHTTPResult[2][3] > GVL_Const.cISOClassDef_Displ[intMachineSelected, intElasticitySelected, 1] THEN
            ISOClassIs_Displ := E_IsoClass.B;
        END_IF;

        // according to ISO 10816-3 select worst case 		
        ISO_10816_Classification := E_IsoClass.A;

        IF ISOClassIs_Vel > ISO_10816_Classification THEN
            ISO_10816_Classification := ISOClassIs_Vel;
        END_IF

        IF ISOClassIs_Displ > ISO_10816_Classification THEN
            ISO_10816_Classification := ISOClassIs_Displ;
        END_IF

    ELSE
        // result is NaN... code here what to do. 

    END_IF;

END_IF
END_ACTION

ACTION SinkData:
(* Push results to sink *)
fbSinkISO.Output2DStd(pDataOut     := ADR(GLOBAL.aSensorWorkISOHTTPResult[2]),
                      nDataOutSize := SIZEOF(GLOBAL.aSensorWorkISOHTTPResult[2]),
                      eElementType := eMA_TypeCode_LREAL,
                      nOptionPars  := 0,

                      bNewResult => bCalculateISO);

IF fbSinkISO.bError THEN
    fbErrHist.AddError(bErr := TRUE, hrErrCode := fbSinkISO.hrErrorCode, sErrSource := 'CM_SensorWorks_Sensor2.fbSinkISO'); // error monitoring
    // ToDo: if error
END_IF
END_ACTION

ACTION SourceData:

IF GLOBAL.stSensorWorksHTTPSensorData[2].timestamp <> strOldTS THEN
    FOR i := 1 TO GVL_Const.cSensorPacket DO
        GLOBAL.aSensorWorksHTTPInput[2][i] := GLOBAL.stSensorWorksHTTPSensorData[2].value[i] * GLOBAL.stSensorWorksHTTPSensorData[2].calibration;
    END_FOR

    bNewSensorDataAvailable := TRUE;
END_IF

// Collection
IF bNewSensorDataAvailable THEN
    // Check to make sure code works
    (*	
	testwave(
	
			bEnable:= TRUE, 
			fFrequency 	:= testfq,
			fAmplitude 	:= 100,
			eFunction 	:= E_FunctionType.Sine,
			aSignal		:= GLOBAL.aSensorWorksHTTPInput[1]);	
	// end of signal generation
*)

    fbSource_SensorWorks.Input2DStd(pDataIn      := ADR(GLOBAL.aSensorWorksHTTPInput[2]),
                                    nDataInSize  := SIZEOF(GLOBAL.aSensorWorksHTTPInput[2]),
                                    eElementType := eMA_TypeCode_LREAL,
                                    nOptionPars  := Tc3_CM.cCMA_Option_MarkInterruption);

    bNewSensorDataAvailable := FALSE; // reset flag
    //testwave.bEnable := FALSE;
END_IF

// Check for errors
IF fbSource_SensorWorks.bError THEN
    fbErrHist.AddError(bErr := TRUE, hrErrCode := fbSource_SensorWorks.hrErrorCode, sErrSource := 'CM_SensorWorks_Sensor2.SourceData');
END_IF

strOldTS := GLOBAL.stSensorWorksHTTPSensorData[2].timestamp;
END_ACTION

END_PROGRAM

// ---- FUBs/FB_Flash.TcPOU
FUNCTION_BLOCK FB_Flash
VAR_INPUT
	Input : ARRAY[0..999] OF BOOL;
	OffTime : TIME;
	OnTime :  TIME;
END_VAR
VAR_OUTPUT
	Output : ARRAY[0..999] OF BOOL;
END_VAR
VAR
	OffTimer : TON;
	OnTimer	:	TON;
	i: INT;
END_VAR

OnTimer.PT 	:= OnTime;
OffTimer.PT := OffTime;

OffTimer.IN := NOT(OnTimer.Q);
OnTimer.IN := OffTimer.Q;
		
	
FOR i := 0 TO 999 DO
	IF Input[i] THEN
		Output[i] := OnTimer.IN;
	ELSE 
		Output[i] := FALSE;
	END_IF
END_FOR
OnTimer();
OffTimer();

END_FUNCTION_BLOCK
